// Mitsubishi GX Works2 project: ハウステンボス用   PLC: Q03UDV

PROGRAM MAIN
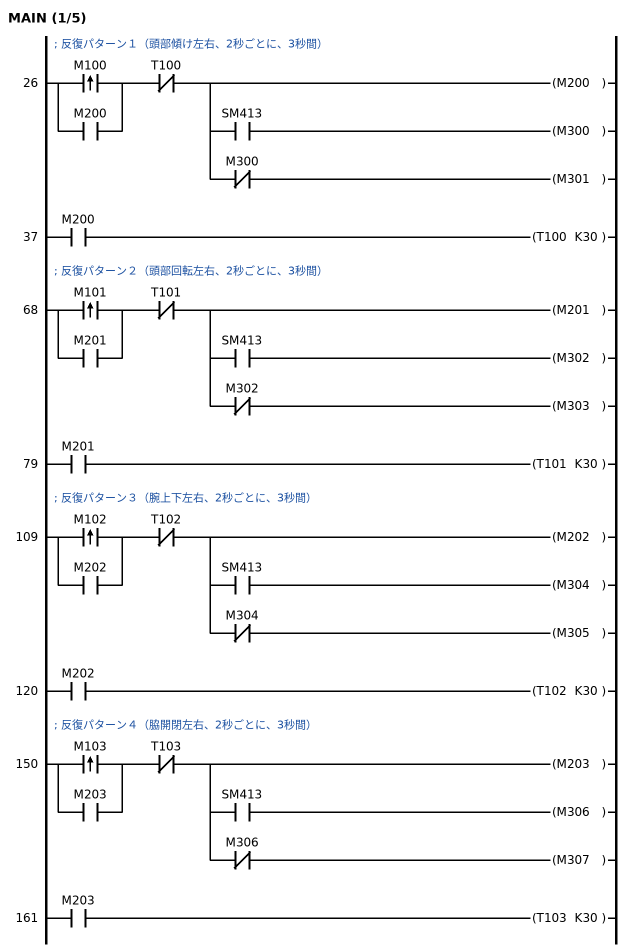
; 反復パターン１（頭部傾け左右、2秒ごとに、3秒間）
26    LDP     M100
      OR      M200
      ANI     T100
      OUT     M200
      MPS
      AND     SM413
      OUT     M300
      MPP
      ANI     M300
      OUT     M301
37    LD      M200
      OUT     T100 K30
; 反復パターン２（頭部回転左右、2秒ごとに、3秒間）
68    LDP     M101
      OR      M201
      ANI     T101
      OUT     M201
      MPS
      AND     SM413
      OUT     M302
      MPP
      ANI     M302
      OUT     M303
79    LD      M201
      OUT     T101 K30
; 反復パターン３（腕上下左右、2秒ごとに、3秒間）
109   LDP     M102
      OR      M202
      ANI     T102
      OUT     M202
      MPS
      AND     SM413
      OUT     M304
      MPP
      ANI     M304
      OUT     M305
120   LD      M202
      OUT     T102 K30
; 反復パターン４（脇開閉左右、2秒ごとに、3秒間）
150   LDP     M103
      OR      M203
      ANI     T103
      OUT     M203
      MPS
      AND     SM413
      OUT     M306
      MPP
      ANI     M306
      OUT     M307
161   LD      M203
      OUT     T103 K30
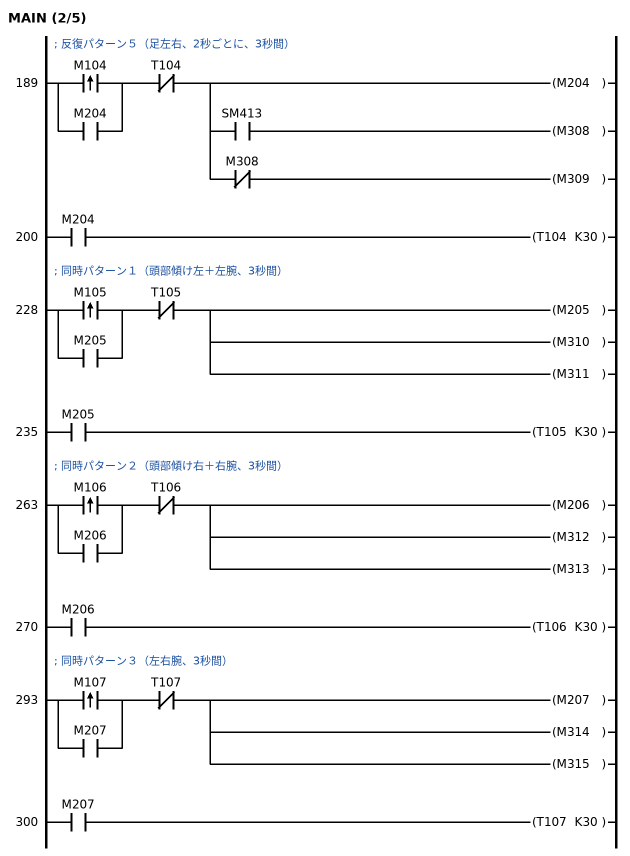
; 反復パターン５（足左右、2秒ごとに、3秒間）
189   LDP     M104
      OR      M204
      ANI     T104
      OUT     M204
      MPS
      AND     SM413
      OUT     M308
      MPP
      ANI     M308
      OUT     M309
200   LD      M204
      OUT     T104 K30
; 同時パターン１（頭部傾け左＋左腕、3秒間）
228   LDP     M105
      OR      M205
      ANI     T105
      OUT     M205
      OUT     M310
      OUT     M311
235   LD      M205
      OUT     T105 K30
; 同時パターン２（頭部傾け右＋右腕、3秒間）
263   LDP     M106
      OR      M206
      ANI     T106
      OUT     M206
      OUT     M312
      OUT     M313
270   LD      M206
      OUT     T106 K30
; 同時パターン３（左右腕、3秒間）
293   LDP     M107
      OR      M207
      ANI     T107
      OUT     M207
      OUT     M314
      OUT     M315
300   LD      M207
      OUT     T107 K30
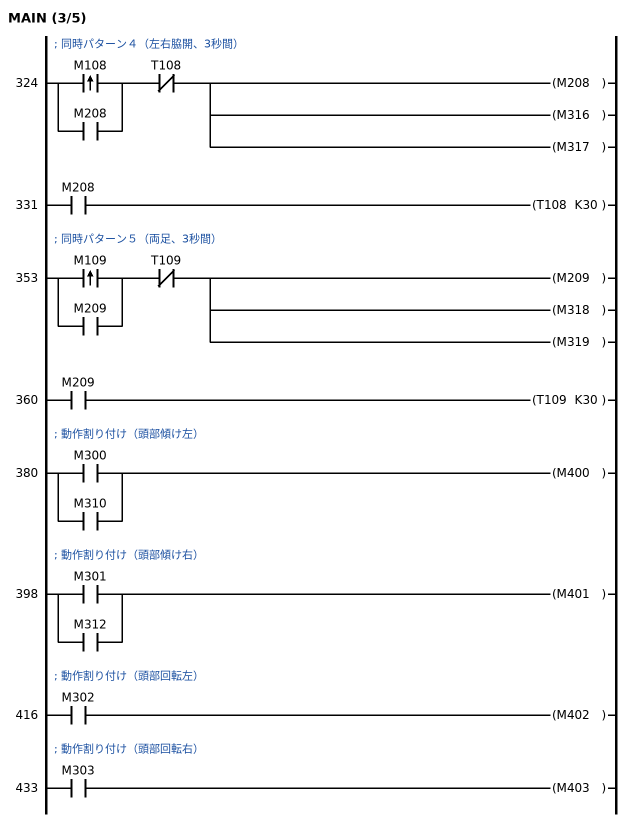
; 同時パターン４（左右脇開、3秒間）
324   LDP     M108
      OR      M208
      ANI     T108
      OUT     M208
      OUT     M316
      OUT     M317
331   LD      M208
      OUT     T108 K30
; 同時パターン５（両足、3秒間）
353   LDP     M109
      OR      M209
      ANI     T109
      OUT     M209
      OUT     M318
      OUT     M319
360   LD      M209
      OUT     T109 K30
; 動作割り付け（頭部傾け左）
380   LD      M300
      OR      M310
      OUT     M400
; 動作割り付け（頭部傾け右）
398   LD      M301
      OR      M312
      OUT     M401
; 動作割り付け（頭部回転左）
416   LD      M302
      OUT     M402
; 動作割り付け（頭部回転右）
433   LD      M303
      OUT     M403
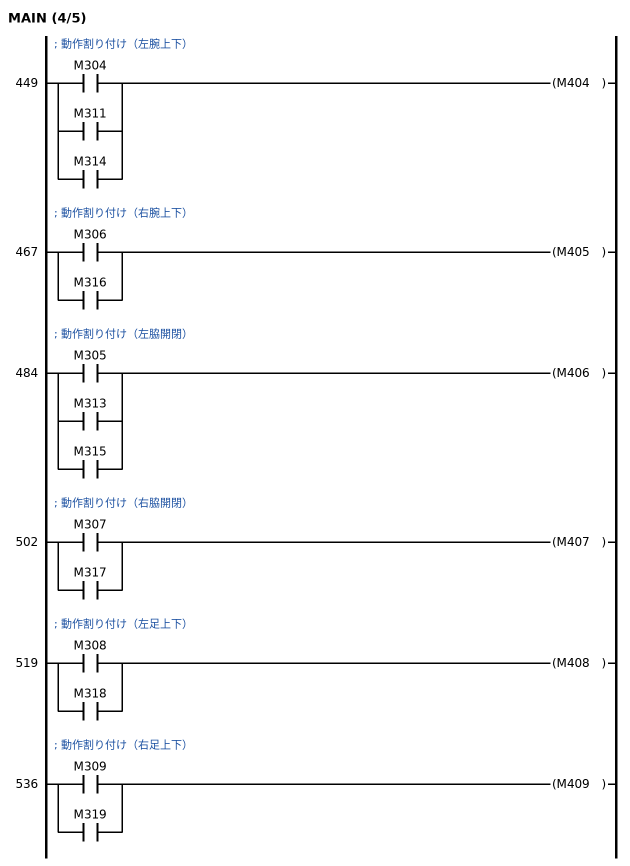
; 動作割り付け（左腕上下）
449   LD      M304
      OR      M311
      OR      M314
      OUT     M404
; 動作割り付け（右腕上下）
467   LD      M306
      OR      M316
      OUT     M405
; 動作割り付け（左脇開閉）
484   LD      M305
      OR      M313
      OR      M315
      OUT     M406
; 動作割り付け（右脇開閉）
502   LD      M307
      OR      M317
      OUT     M407
; 動作割り付け（左足上下）
519   LD      M308
      OR      M318
      OUT     M408
; 動作割り付け（右足上下）
536   LD      M309
      OR      M319
      OUT     M409
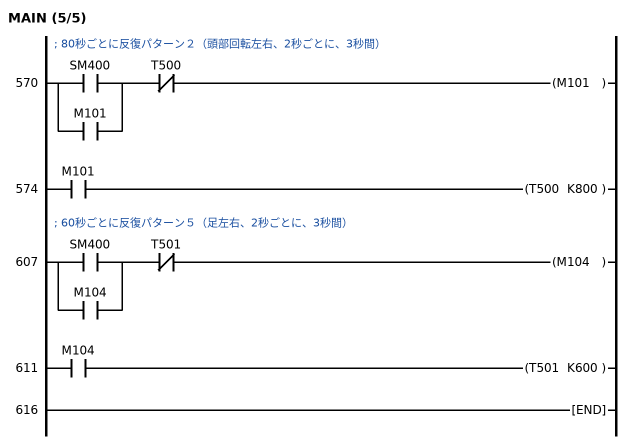
; 80秒ごとに反復パターン２（頭部回転左右、2秒ごとに、3秒間）
570   LD      SM400
      OR      M101
      ANI     T500
      OUT     M101
574   LD      M101
      OUT     T500 K800
; 60秒ごとに反復パターン５（足左右、2秒ごとに、3秒間）
607   LD      SM400
      OR      M104
      ANI     T501
      OUT     M104
611   LD      M104
      OUT     T501 K600
616   END
END_PROGRAM
